// TIA Portal V16 export
// export: Created 2021-08-30T11:09:31.9984935Z, ExportSetting WithDefaults, DisplayName Totally Integrated Automation Portal, DisplayVersion V16 Update 3, DisplayName TIA Portal Version Control Interface, DisplayVersion V16 Update 2, DisplayName TIA Portal Openness, DisplayVersion V16 Update 3, DisplayName TIA Portal Teamcenter Gateway, DisplayVersion V16, DisplayName STEP 7 Professional, DisplayVersion V16 Update 3, DisplayName STEP 7 Safety, DisplayVersion V16, DisplayName WinCC Advanced, DisplayVersion V16 Update 3
FUNCTION_BLOCK "PID_Pump2Pu1Fc"   // FB59, FBD
{ S7_Optimized_Access := 'TRUE' }
VERSION : 0.1
// stored: AutoNumber true, IsIECCheckEnabled false, IsRetainMemResEnabled false, MemoryReserve 100, SetENOAutomatically false, UDAEnableTagReadback false
   VAR_INPUT
      value : Real;
      PU1 : "Pump";
      PU2 : "Pump";
   END_VAR
   VAR_OUTPUT
      outPER : Int;
   END_VAR
   VAR_IN_OUT
      pidSet : "setPID";
      PID_Compact : PID_Compact;
   END_VAR
   VAR
      pTrigAutoMode : Bool;
      pTrigManualMode : Bool;
      pTrigCmAuto1 : Bool;
      pTrigCmAuto2 : Bool;
      nTrigCmAuto1 : Bool;
      nTrigCmAuto2 : Bool;
      pTrigFix : Bool;
      nTrigFix : Bool;
      pTrigFreez : Bool;
      nTrigFreez : Bool;
      pTrigCmHand : Bool;
      nTrigCmHand : Bool;
   END_VAR
   VAR_TEMP   // added for the SCL form of the ladder/FBD networks
      _w1 : Bool;
      _w2 : Bool;
      _w3 : Bool;
      _w4 : Bool;
      _w5 : Bool;
      _w6 : Bool;
      _w7 : Bool;
      _w8 : Bool;
      _w9 : Bool;
      _w10 : Bool;
   END_VAR
BEGIN

REGION Network 1: Интеграл
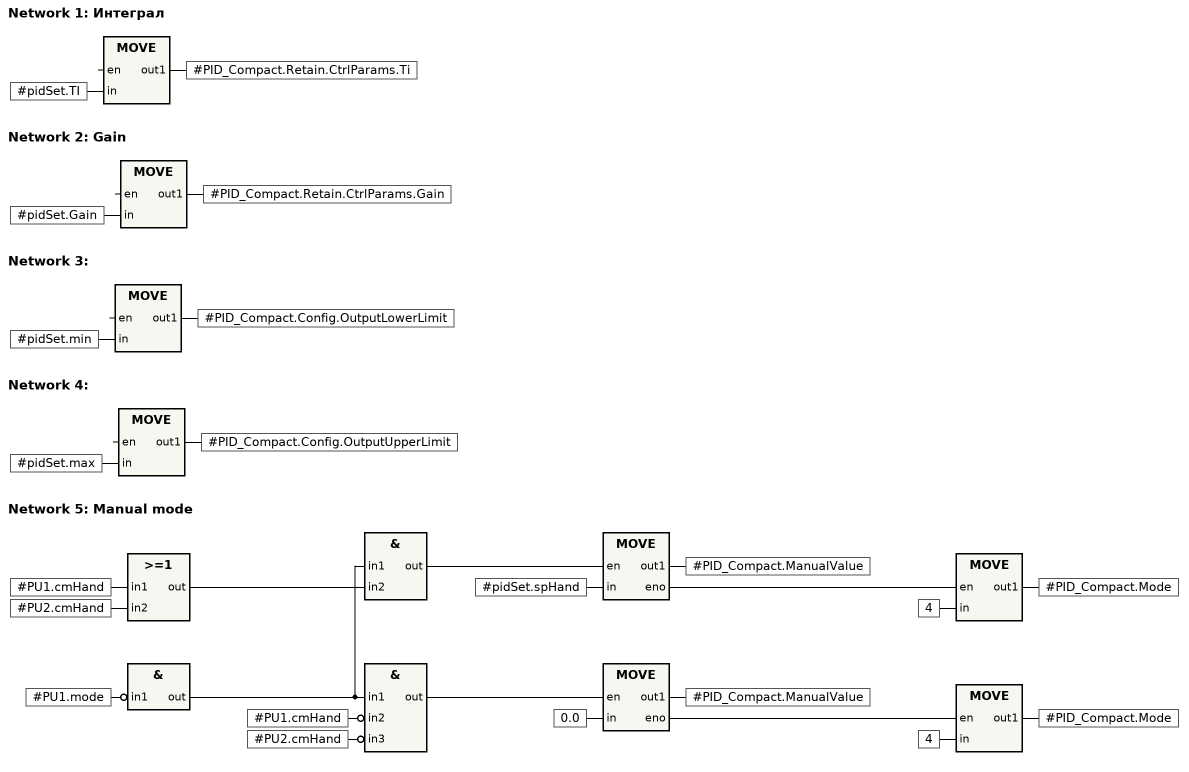
   #PID_Compact.Retain.CtrlParams.Ti := #pidSet.TI;
END_REGION

REGION Network 2: Gain
   #PID_Compact.Retain.CtrlParams.Gain := #pidSet.Gain;
END_REGION

REGION Network 3
   #PID_Compact.Config.OutputLowerLimit := #pidSet.min;
END_REGION

REGION Network 4
   #PID_Compact.Config.OutputUpperLimit := #pidSet.max;
END_REGION

REGION Network 5: Manual mode
   IF NOT #PU1.mode AND (#PU1.cmHand OR #PU2.cmHand) THEN
       #PID_Compact.ManualValue := #pidSet.spHand;
       #PID_Compact.Mode := 4;
   END_IF;
   IF NOT #PU1.mode AND NOT #PU1.cmHand AND NOT #PU2.cmHand THEN
       #PID_Compact.ManualValue := 0.0;
       #PID_Compact.Mode := 4;
   END_IF;
END_REGION

REGION Network 6: Auto mode
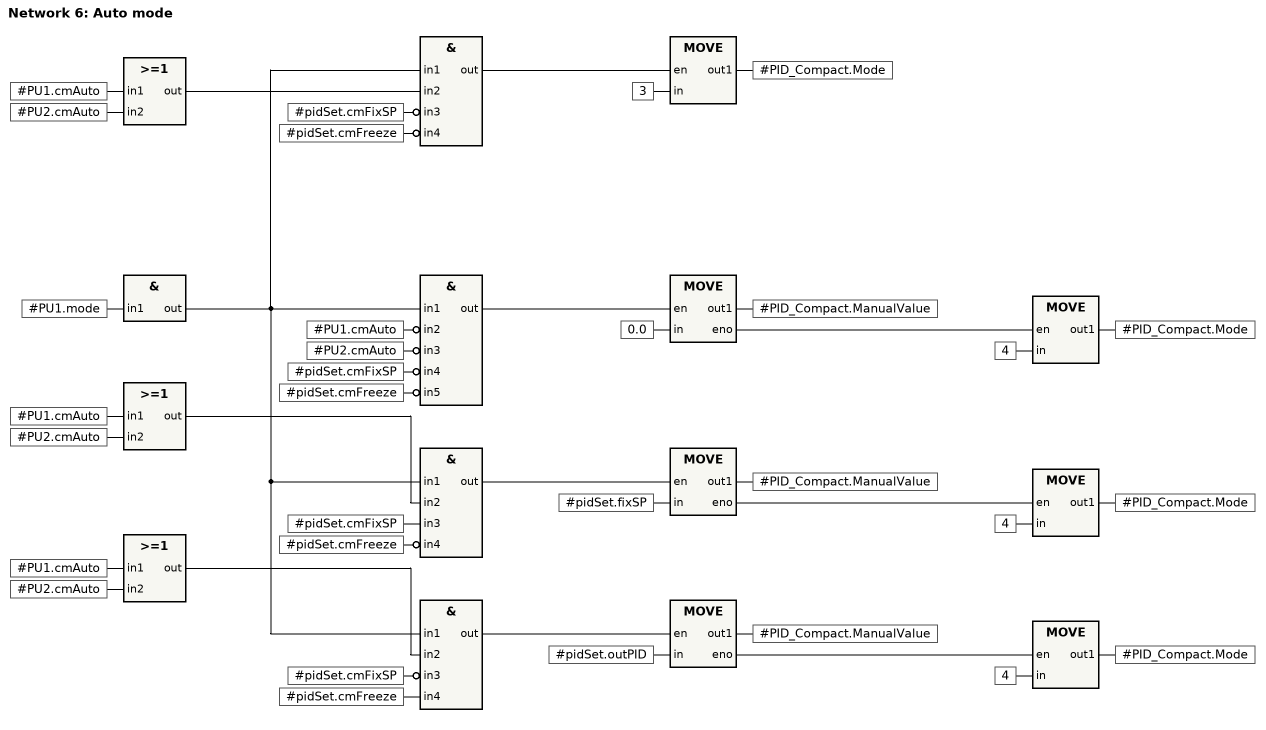
   IF #PU1.mode AND (#PU1.cmAuto OR #PU2.cmAuto) AND NOT #pidSet.cmFixSP AND NOT #pidSet.cmFreeze THEN
       #PID_Compact.Mode := 3;
   END_IF;
   IF #PU1.mode AND NOT #PU1.cmAuto AND NOT #PU2.cmAuto AND NOT #pidSet.cmFixSP AND NOT #pidSet.cmFreeze THEN
       #PID_Compact.ManualValue := 0.0;
       #PID_Compact.Mode := 4;
   END_IF;
   IF #PU1.mode AND (#PU1.cmAuto OR #PU2.cmAuto) AND #pidSet.cmFixSP AND NOT #pidSet.cmFreeze THEN
       #PID_Compact.ManualValue := #pidSet.fixSP;
       #PID_Compact.Mode := 4;
   END_IF;
   IF #PU1.mode AND (#PU1.cmAuto OR #PU2.cmAuto) AND NOT #pidSet.cmFixSP AND #pidSet.cmFreeze THEN
       #PID_Compact.ManualValue := #pidSet.outPID;
       #PID_Compact.Mode := 4;
   END_IF;
END_REGION

REGION Network 7: Set modeActivate
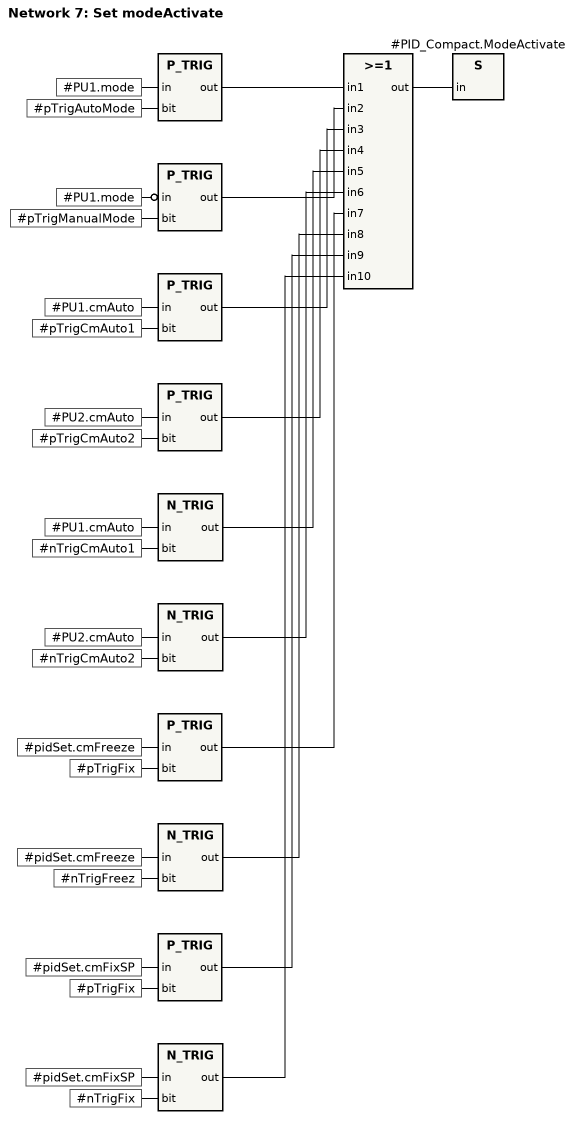
   #_w1 := #PU1.mode AND NOT #pTrigAutoMode;   // rising edge
   #pTrigAutoMode := #PU1.mode;
   #_w2 := NOT #PU1.mode AND NOT #pTrigManualMode;   // rising edge
   #pTrigManualMode := NOT #PU1.mode;
   #_w3 := #PU1.cmAuto AND NOT #pTrigCmAuto1;   // rising edge
   #pTrigCmAuto1 := #PU1.cmAuto;
   #_w4 := #PU2.cmAuto AND NOT #pTrigCmAuto2;   // rising edge
   #pTrigCmAuto2 := #PU2.cmAuto;
   #_w5 := NOT #PU1.cmAuto AND #nTrigCmAuto1;   // falling edge
   #nTrigCmAuto1 := #PU1.cmAuto;
   #_w6 := NOT #PU2.cmAuto AND #nTrigCmAuto2;   // falling edge
   #nTrigCmAuto2 := #PU2.cmAuto;
   #_w7 := #pidSet.cmFreeze AND NOT #pTrigFix;   // rising edge
   #pTrigFix := #pidSet.cmFreeze;
   #_w8 := NOT #pidSet.cmFreeze AND #nTrigFreez;   // falling edge
   #nTrigFreez := #pidSet.cmFreeze;
   #_w9 := #pidSet.cmFixSP AND NOT #pTrigFix;   // rising edge
   #pTrigFix := #pidSet.cmFixSP;
   #_w10 := NOT #pidSet.cmFixSP AND #nTrigFix;   // falling edge
   #nTrigFix := #pidSet.cmFixSP;
   IF #_w1 OR #_w2 OR #_w3 OR #_w4 OR #_w5 OR #_w6 OR #_w7 OR #_w8 OR #_w9 OR #_w10 THEN
       #PID_Compact.ModeActivate := TRUE;
   END_IF;
END_REGION

REGION Network 8
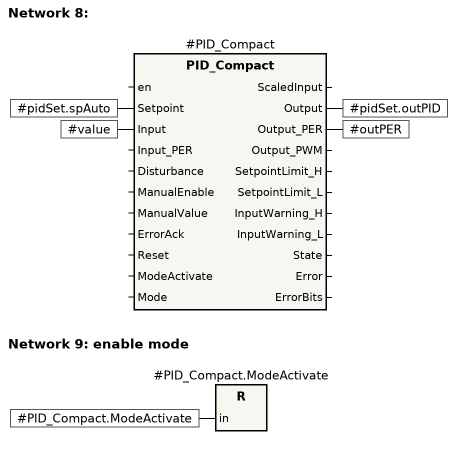
   #PID_Compact(Setpoint := #pidSet.spAuto, Input := #value, Output => #pidSet.outPID, Output_PER => #outPER);   // PID_Compact
END_REGION

REGION Network 9: enable mode
   IF #PID_Compact.ModeActivate THEN #PID_Compact.ModeActivate := FALSE; END_IF;
END_REGION
END_FUNCTION_BLOCK
